// TIA Portal project "Foerderband" (V18)

(* hardware
DEVICE "S7-1500/ET200MP-Station_1"  S7-1500 station
   slot 0: "Profilschiene_0"  Rack  6ES7 590-1***0-0AA0
   slot 1: "Rohlager01SPS"  CPU 1516-3 PN/DP  6ES7 516-3AN01-0AB0  V2.6
      slot 3: "CPU-Display_1"  6ES7591-1BA00-0AA0
      slot 32768: "PROFINET-Schnittstelle_1"  X1
         slot 32769: "Port_1"  X1 P1
         slot 32770: "Port_2"  X1 P2
      slot 33024: "PROFINET-Schnittstelle_2"  X2
         slot 33025: "Port_1"  X2 P1
      slot 33280: "DP-Schnittstelle_1"  X3
   slot 2: "AI 8xU/I/RTD/TC ST_1"  AI 8xU/I/RTD/TC ST  6ES7 531-7KF00-0AB0  V2.0
   slot 3: "AQ 4xU/I ST_1"  AQ 4xU/I ST  6ES7 532-5HD00-0AB0  V2.0
   slot 4: "DI 32x24VDC HF_1"  DI 32x24VDC HF  6ES7 521-1BL00-0AB0  V2.1
   slot 5: "DQ 32x24VDC/0.5A HF_1"  DQ 32x24VDC/0.5A HF  6ES7 522-1BL01-0AB0  V1.0
DEVICE "ET 200SP-Station_1"  ET 200SP-Station
   slot 0: "Baugruppenträger_0"  Rack  6ES5 710-8MAx1
   slot 0: "Rohlager01DP"  IM 155-6 PN HF  6ES7 155-6AU00-0CN0  V3.3
   slot 1: "DI 8x24VDC HF_1"  DI 8x24VDC HF  6ES7 131-6BF00-0CA0  V2.0
      slot 1: "DI 8x24VDC HF_1"  DI 8x24VDC HF
   slot 2: "DQ 8x24VDC/0.5A HF_1"  DQ 8x24VDC/0.5A HF  6ES7 132-6BF00-0CA0  V2.0
      slot 1: "DQ 8x24VDC/0.5A HF_1"  DQ 8x24VDC/0.5A HF
   slot 3: "DI 8x24VDC HF_2"  DI 8x24VDC HF  6ES7 131-6BF00-0CA0  V2.0
      slot 1: "DI 8x24VDC HF_2"  DI 8x24VDC HF
   slot 4: "DQ 8x24VDC/0.5A HF_2"  DQ 8x24VDC/0.5A HF  6ES7 132-6BF00-0CA0  V2.0
      slot 1: "DQ 8x24VDC/0.5A HF_2"  DQ 8x24VDC/0.5A HF
   slot 5: "CM 4xIO-Link_1"  CM 4xIO-Link  6ES7 137-6BD00-0BA0  V2.1
      slot 1: "CM 4xIO-Link_1"  6ES7 137-6BD00-0BA0
   slot 6: "Servermodul_1"  Server module  6ES7 193-6PA00-0AA0  V1.1
      slot 1: "Servermodul_1"  Server module
   slot 127: "BA 2xRJ45"  BA 2xRJ45  6ES7 193-6AR00-0AA0  V0.0
      slot 1: "Port_1"  X1 P1 R  6ES7 193-6AR00-0AA0  V0.0
      slot 2: "Port_2"  X1 P2 R  6ES7 193-6AR00-0AA0  V0.0
*)

// ===== PLC "Rohlager01SPS"  CPU 1516-3 PN/DP =====

VAR_GLOBAL   // PLC tag table "Standard-Variablentabelle"
   "System_Byte" AT %MB1 : Byte;
   "FirstScan" AT %M1.0 : Bool;
   "DiagStatusUpdate" AT %M1.1 : Bool;
   "AlwaysTRUE" AT %M1.2 : Bool;
   "AlwaysFALSE" AT %M1.3 : Bool;
   "BG1_Conveyor_sensor_left" AT %I50.0 : Bool;
   "BG2_Conveyor_sensor_rigth" AT %I50.1 : Bool;
   "BG1_Position Left" AT %I51.0 : Bool;
   "BG4_Stopper Rigth" AT %I51.3 : Bool;
   "BG6_Plunger_Bottom" AT %I51.5 : Bool;
   "BG7_Plunger_Middle" AT %I51.6 : Bool;
   "BG8_Plunger_Top" AT %I51.7 : Bool;
   "Q_Motor_Clockwise rotation" AT %Q50.6 : Bool;
   "Q_Separator" AT %Q51.2 : Bool;
   "Q_Plunger up" AT %Q51.3 : Bool;
   "Q_Plunger Down" AT %Q51.4 : Bool;
   "Clock_Byte" AT %MB0 : Byte;
   "Clock_10Hz" AT %M0.0 : Bool;
   "Clock_5Hz" AT %M0.1 : Bool;
   "Clock_2.5Hz" AT %M0.2 : Bool;
   "Clock_2Hz" AT %M0.3 : Bool;
   "Clock_1.25Hz" AT %M0.4 : Bool;
   "Clock_1Hz" AT %M0.5 : Bool;
   "Clock_0.625Hz" AT %M0.6 : Bool;
   "Clock_0.5Hz" AT %M0.7 : Bool;
   "BG2_Position Rigth" AT %I51.1 : Bool;
END_VAR

DATA_BLOCK "System_DB"   // DB1
{ S7_Optimized_Access := 'TRUE' }
VERSION : 0.1
// stored: InstanceOfName System
"System"
BEGIN
END_DATA_BLOCK

FUNCTION_BLOCK "Sequencer"   // FB1, FBD
{ S7_Optimized_Access := 'TRUE' }
VERSION : 0.1
   VAR_INPUT
      BG1_Conveyor_sensor_left : Bool;
      BG2_Conveyor_sensor_rigth : Bool;
      BG6_Plunger_Bottom : Bool;
      BG7_Plunger_Middle : Bool;
      BG8_Plunger_Top : Bool;
      "BG1_Position Left" : Bool;
      "BG2_Position Rigth" : Bool;
      FirstScan : Bool;
   END_VAR
   VAR
      Step_0 : Bool;
      Step_1 : Bool;
      Step_2 : Bool;
      Step_3 : Bool;
      Step_4 : Bool;
      Step_5 : Bool;
      Step_6 : Bool;
      Step_7 : Bool;
      Step_8 : Bool;
      Step_9 : Bool;
   END_VAR
BEGIN

REGION Network 1: X_0
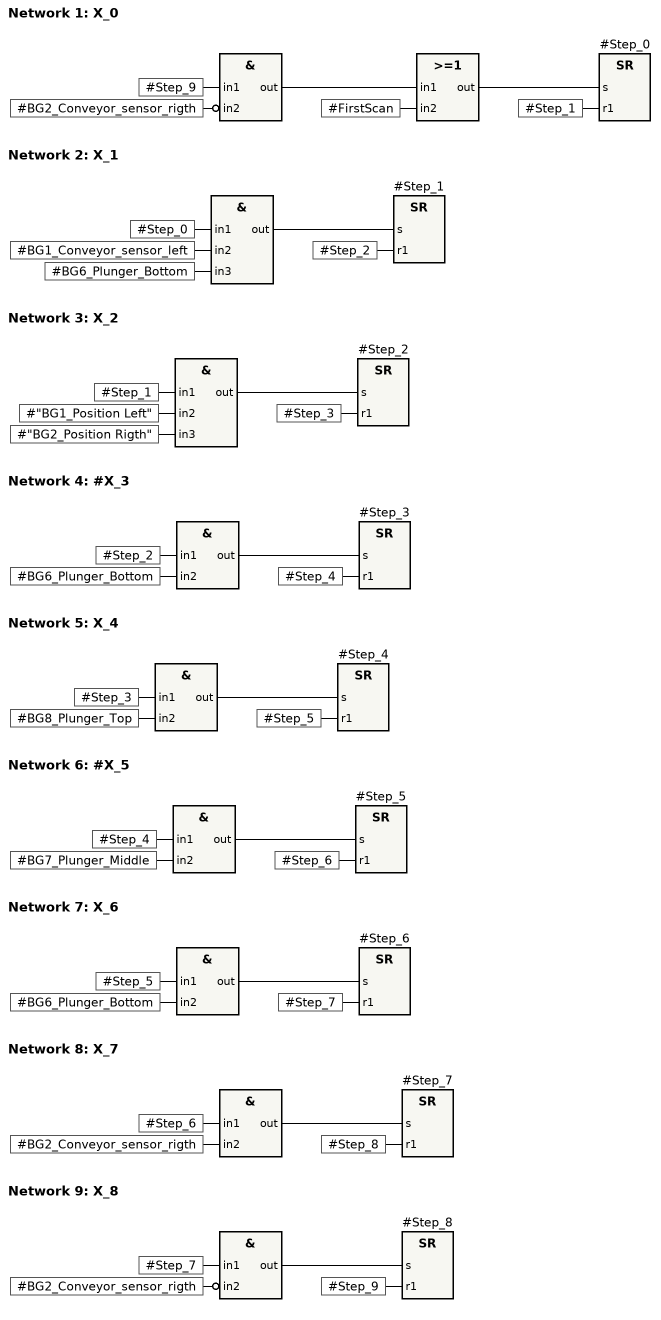
   IF (#Step_9 AND NOT #BG2_Conveyor_sensor_rigth) OR #FirstScan THEN
       #Step_0 := TRUE;   // SR flip-flop
   END_IF;
   IF #Step_1 THEN #Step_0 := FALSE; END_IF;
END_REGION

REGION Network 2: X_1
   IF #Step_0 AND #BG1_Conveyor_sensor_left AND #BG6_Plunger_Bottom THEN
       #Step_1 := TRUE;   // SR flip-flop
   END_IF;
   IF #Step_2 THEN #Step_1 := FALSE; END_IF;
END_REGION

REGION Network 3: X_2
   IF #Step_1 AND #"BG1_Position Left" AND #"BG2_Position Rigth" THEN
       #Step_2 := TRUE;   // SR flip-flop
   END_IF;
   IF #Step_3 THEN #Step_2 := FALSE; END_IF;
END_REGION

REGION Network 4: #X_3
   IF #Step_2 AND #BG6_Plunger_Bottom THEN
       #Step_3 := TRUE;   // SR flip-flop
   END_IF;
   IF #Step_4 THEN #Step_3 := FALSE; END_IF;
END_REGION

REGION Network 5: X_4
   IF #Step_3 AND #BG8_Plunger_Top THEN
       #Step_4 := TRUE;   // SR flip-flop
   END_IF;
   IF #Step_5 THEN #Step_4 := FALSE; END_IF;
END_REGION

REGION Network 6: #X_5
   IF #Step_4 AND #BG7_Plunger_Middle THEN
       #Step_5 := TRUE;   // SR flip-flop
   END_IF;
   IF #Step_6 THEN #Step_5 := FALSE; END_IF;
END_REGION

REGION Network 7: X_6
   IF #Step_5 AND #BG6_Plunger_Bottom THEN
       #Step_6 := TRUE;   // SR flip-flop
   END_IF;
   IF #Step_7 THEN #Step_6 := FALSE; END_IF;
END_REGION

REGION Network 8: X_7
   IF #Step_6 AND #BG2_Conveyor_sensor_rigth THEN
       #Step_7 := TRUE;   // SR flip-flop
   END_IF;
   IF #Step_8 THEN #Step_7 := FALSE; END_IF;
END_REGION

REGION Network 9: X_8
   IF #Step_7 AND NOT #BG2_Conveyor_sensor_rigth THEN
       #Step_8 := TRUE;   // SR flip-flop
   END_IF;
   IF #Step_9 THEN #Step_8 := FALSE; END_IF;
END_REGION

REGION Network 10: X_9
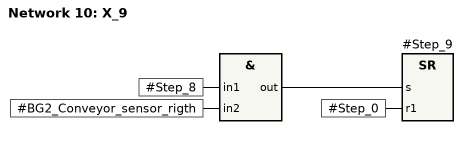
   IF #Step_8 AND #BG2_Conveyor_sensor_rigth THEN
       #Step_9 := TRUE;   // SR flip-flop
   END_IF;
   IF #Step_0 THEN #Step_9 := FALSE; END_IF;
END_REGION
END_FUNCTION_BLOCK

FUNCTION_BLOCK "Outputs"   // FB2, FBD
{ S7_Optimized_Access := 'TRUE' }
VERSION : 0.1
   VAR_INPUT
      Step_0 : Bool;
      Step_1 : Bool;
      Step_2 : Bool;
      Step_3 : Bool;
      Step_4 : Bool;
      Step_5 : Bool;
      Step_6 : Bool;
      Step_7 : Bool;
      Step_8 : Bool;
      Step_9 : Bool;
   END_VAR
   VAR_OUTPUT
      Conveyor : Bool;
      Separator : Bool;
      Plunger_Up : Bool;
      Plunger_Down : Bool;
   END_VAR
BEGIN

REGION Network 1: Band_2
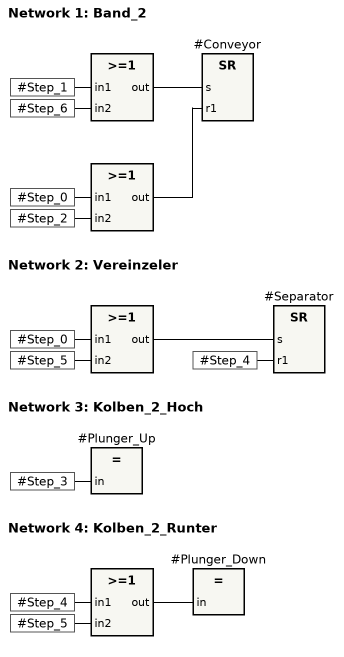
   IF #Step_1 OR #Step_6 THEN
       #Conveyor := TRUE;   // SR flip-flop
   END_IF;
   IF #Step_0 OR #Step_2 THEN #Conveyor := FALSE; END_IF;
END_REGION

REGION Network 2: Vereinzeler
   IF #Step_0 OR #Step_5 THEN
       #Separator := TRUE;   // SR flip-flop
   END_IF;
   IF #Step_4 THEN #Separator := FALSE; END_IF;
END_REGION

REGION Network 3: Kolben_2_Hoch
   #Plunger_Up := #Step_3;
END_REGION

REGION Network 4: Kolben_2_Runter
   #Plunger_Down := #Step_4 OR #Step_5;
END_REGION
END_FUNCTION_BLOCK

FUNCTION_BLOCK "System"   // FB3, FBD
{ S7_Optimized_Access := 'TRUE' }
VERSION : 0.1
   VAR_INPUT
      BG1_Conveyor_sensor_left : Bool;
      BG2_Conveyor_sensor_rigth : Bool;
      "BG1_Position Left" : Bool;
      "BG4_Stopper Rigth" : Bool;
      BG6_Plunger_Bottom : Bool;
      BG7_Plunger_Middle : Bool;
      BG8_Plunger_Top : Bool;
      FirstScan : Bool;
   END_VAR
   VAR_OUTPUT
      Motor_Conveyor : Bool;
      Separator : Bool;
      "Plunger Up" : Bool;
      "Plunger Down" : Bool;
   END_VAR
   VAR
      Sequencer_Instance : "Sequencer";
      Outputs_Instance : "Outputs";
   END_VAR
BEGIN

REGION Network 1: Schrittkette
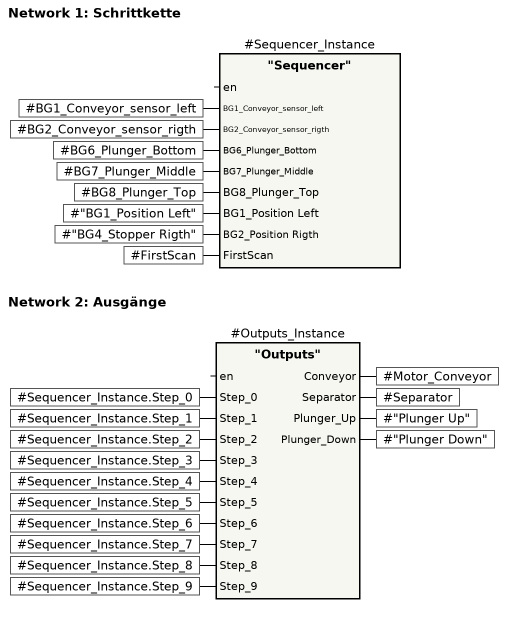
   #Sequencer_Instance(BG1_Conveyor_sensor_left := #BG1_Conveyor_sensor_left,   // "Sequencer"
                       BG2_Conveyor_sensor_rigth := #BG2_Conveyor_sensor_rigth,
                       BG6_Plunger_Bottom := #BG6_Plunger_Bottom,
                       BG7_Plunger_Middle := #BG7_Plunger_Middle,
                       BG8_Plunger_Top := #BG8_Plunger_Top,
                       "BG1_Position Left" := #"BG1_Position Left",
                       "BG2_Position Rigth" := #"BG4_Stopper Rigth",
                       FirstScan := #FirstScan);
END_REGION

REGION Network 2: Ausgänge
   #Outputs_Instance(Step_0 := #Sequencer_Instance.Step_0,   // "Outputs"
                     Step_1 := #Sequencer_Instance.Step_1,
                     Step_2 := #Sequencer_Instance.Step_2,
                     Step_3 := #Sequencer_Instance.Step_3,
                     Step_4 := #Sequencer_Instance.Step_4,
                     Step_5 := #Sequencer_Instance.Step_5,
                     Step_6 := #Sequencer_Instance.Step_6,
                     Step_7 := #Sequencer_Instance.Step_7,
                     Step_8 := #Sequencer_Instance.Step_8,
                     Step_9 := #Sequencer_Instance.Step_9,
                     Conveyor => #Motor_Conveyor,
                     Separator => #Separator,
                     Plunger_Up => #"Plunger Up",
                     Plunger_Down => #"Plunger Down");
END_REGION
END_FUNCTION_BLOCK

ORGANIZATION_BLOCK "Main"   // OB1, FBD, ProgramCycle
TITLE = "Main Program Sweep (Cycle)"
{ S7_Optimized_Access := 'TRUE' }
VERSION : 0.1
   VAR_INPUT
      Initial_Call : Bool;   // Initial call of this OB
      Remanence : Bool;   // =True, if remanent data are available
   END_VAR
BEGIN

REGION Network 1
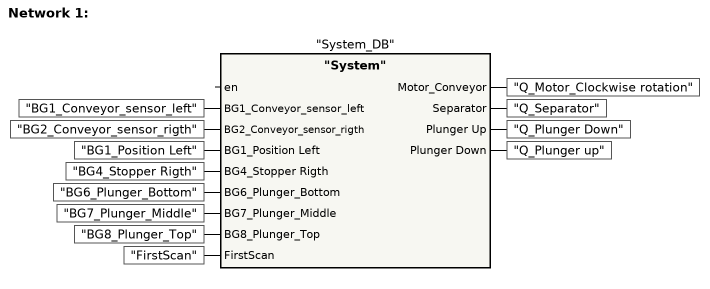
   "System_DB"(BG1_Conveyor_sensor_left := "BG1_Conveyor_sensor_left",   // "System"
               BG2_Conveyor_sensor_rigth := "BG2_Conveyor_sensor_rigth",
               "BG1_Position Left" := "BG1_Position Left",
               "BG4_Stopper Rigth" := "BG4_Stopper Rigth",
               BG6_Plunger_Bottom := "BG6_Plunger_Bottom",
               BG7_Plunger_Middle := "BG7_Plunger_Middle",
               BG8_Plunger_Top := "BG8_Plunger_Top",
               FirstScan := "FirstScan",
               Motor_Conveyor => "Q_Motor_Clockwise rotation",
               Separator => "Q_Separator",
               "Plunger Up" => "Q_Plunger Down",
               "Plunger Down" => "Q_Plunger up");
END_REGION
END_ORGANIZATION_BLOCK